// TIA Portal project "PLC_Progetto1" (V15)

(* hardware
DEVICE "S7-1200 station_1"  S7-1200 Station
   slot 0: "Rack_0"  S7-1200 Rack  Rack  V1.0
   slot 1: "PLC_1"  CPU 1212C AC/DC/Rly  6ES7 212-1BE40-0XB0  V4.2
   slot 2: "DI 16x24VDC/DQ 16xRelay_1"  SM 1223 DI16/DQ16 x relay  6ES7 223-1PL32-0XB0  V2.0
DEVICE "HMI_1"  KTP700 Basic PN
   slot 0: "HMI_1"  KTP700 Basic PN  6AV2 123-2GB03-0AX0  15.0.0.0
   slot 1: "HMI_RT_1"  KTP700 Basic PN  6AV2 123-2GB03-0AX0  15.0.0.0
   slot 5: "HMI_1.IE_CP_1"  PROFINET Interface  15.0.0.0
      slot 1: "PROFINET Interface_1"  PROFINET Interface
         slot 1: "Port_1"  Port
*)

// ===== PLC "PLC_1"  CPU 1212C AC/DC/Rly =====

VAR_GLOBAL   // PLC tag table "Default tag table"
   "USCITA MA_AVANTI" AT %Q0.0 : Bool;
   "USCITA MA_INDIETRO" AT %Q0.1 : Bool;
   "CAMBIO_VEL" AT %Q0.2 : Bool;
   "Tag_1" AT %IW64 : Word;
END_VAR

DATA_BLOCK "DB"   // DB1
{ S7_Optimized_Access := 'TRUE' }
VERSION : 0.1
   VAR
      MA_AVANTI : Bool;
      MA_INDIETRO : Bool;
      MA_STOP : Bool;
      MA_SPEED : Bool;
      MA_GIRI : Int;
      VAL_INVERTER : Int;
      CALC_2 : Int;
      CALC_3 : Int;
      CALC_4 : Int;
   END_VAR
BEGIN
END_DATA_BLOCK

ORGANIZATION_BLOCK "Main"   // OB1, LAD, ProgramCycle
TITLE = "Main Program Sweep (Cycle)"
{ S7_Optimized_Access := 'TRUE' }
VERSION : 0.1
   VAR_INPUT
      Initial_Call : Bool;   // Initial call of this OB
      Remanence : Bool;   // =True, if remanent data are available
   END_VAR
BEGIN

REGION Network 1
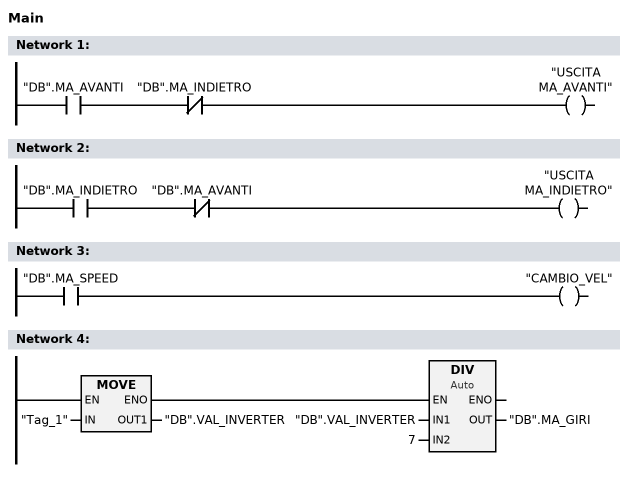
   RUNG wire#powerrail
      Contact( "DB".MA_AVANTI )
      I_Contact( "DB".MA_INDIETRO )
      Coil( "USCITA MA_AVANTI" )
   END_RUNG
   // the same network as SCL:
   "USCITA MA_AVANTI" := "DB".MA_AVANTI AND NOT "DB".MA_INDIETRO;
END_REGION

REGION Network 2
   RUNG wire#powerrail
      Contact( "DB".MA_INDIETRO )
      I_Contact( "DB".MA_AVANTI )
      Coil( "USCITA MA_INDIETRO" )
   END_RUNG
   // the same network as SCL:
   "USCITA MA_INDIETRO" := "DB".MA_INDIETRO AND NOT "DB".MA_AVANTI;
END_REGION

REGION Network 3
   RUNG wire#powerrail
      Contact( "DB".MA_SPEED )
      Coil( "CAMBIO_VEL" )
   END_RUNG
   // the same network as SCL:
   "CAMBIO_VEL" := "DB".MA_SPEED;
END_REGION

REGION Network 4
   RUNG wire#powerrail
      Move(in := "Tag_1", out1 => "DB".VAL_INVERTER)
      Div(in1 := "DB".VAL_INVERTER, in2 := 7, out => "DB".MA_GIRI)
   END_RUNG
   // the same network as SCL:
   "DB".VAL_INVERTER := "Tag_1";
   "DB".MA_GIRI := "DB".VAL_INVERTER / 7;
END_REGION
END_ORGANIZATION_BLOCK

(* ===== HMI "HMI_RT_1" =====
system functions are stored by id; their names below are inferred from use
connection "HMI_Connection_1": ETHERNET, SMART_S7_1200_OMS

HMI tags "Default tag table"
   "DB_MA_GIRI" : Int = PLC "DB".MA_GIRI, 1 s
   "DB_MA_AVANTI" : Bool = PLC "DB".MA_AVANTI, 1 s
   "DB_MA_INDIETRO" : Bool = PLC "DB".MA_INDIETRO, 1 s
   "DB_MA_SPEED" : Bool = PLC "DB".MA_SPEED, 1 s

Template "Template_1" 800x480
   Button "Exit" at 714,429 size 71x50; TextOff 'Exit'; PictureOff "ExitRuntime_KTP700_Basic_PN_TR"; PictureOn "ExitRuntime_KTP700_Basic_PN_TR"
      on Release: StopRuntime(0)
   Button "Template_Button" at 614,429 size 71x50; TextOff 'Text'
   Button "Template_Button_1" at 514,429 size 71x50; TextOff 'Text'
   Button "Template_Button_2" at 414,429 size 71x50; TextOff 'Text'
   Button "Template_Button_3" at 314,429 size 71x50; TextOff 'Text'
   Button "Template_Button_4" at 214,429 size 71x50; TextOff 'Text'
   Button "Template_Button_5" at 114,429 size 71x50; TextOff 'Text'
   Button "Start screen" at 14,429 size 71x50; TextOff 'Start screen'; PictureOff "NavigateHome_KTP700_Basic_PN_TR"; PictureOn "NavigateHome_KTP700_Basic_PN_TR"
      on Release: ActivateScreen("Root screen", 0)

screen "Root screen" 800x480, template "Template_1"
   Button "HmiScreenItemData" at 36,36 size 159x47; TextOff 'Screen0'; PictureOff "Navigates to Screen0 for KTP700 Basic+ PN 15.0.0.0"; PictureOn "Navigates to Screen0 for KTP700 Basic+ PN 15.0.0.0"
      on Release: ActivateScreen("Screen0", 0)

screen "Screen0" 800x480, template "Template_1"
   Button "Back" at 1,1 size 159x47; TextOff 'Back'
      on Release: ActivateScreen("Root screen", 0)
   TextField "Text field_1" at 359,15 size 76x23; Text 'Pagina 0'
   IOField "I/O field_1" at 295,64 size 203x92; FormatPattern 9999
      ProcessValue <- "DB_MA_GIRI"
   Button "Button_1" at 434,167 size 152x50; TextOff 'MARCIA AVANTI'
      on Press: SetBit("DB_MA_AVANTI"); ResetBit("DB_MA_INDIETRO")
   Button "Button_2" at 206,168 size 169x50; TextOff 'MARCIA INDIETRO'
      on Press: SetBit("DB_MA_INDIETRO"); ResetBit("DB_MA_AVANTI")
   Button "Button_3" at 332,253 size 152x50; TextOff 'STOP'
      on Press: ResetBit("DB_MA_AVANTI"); ResetBit("DB_MA_INDIETRO")
   Button "Button_4" at 332,331 size 152x50; TextOff 'VELOCITA''
      on Press: InvertBit("DB_MA_SPEED")
*)